{attribute 'qualified_only'}
{attribute 'strict'}
TYPE yYuklemeBaslatma :
(
	enum_member := 0
);
END_TYPE

(* stored: Version 1.1.0.1, ProductVersion 3.1.4024.12
   DUT yYuklemeBaslatma: Id {e238aabd-79dd-43ec-8e55-5044235f6145} *)
